// TIA Portal V21 export
TYPE "SafetyPLCSignal"
   STRUCT
      "Circuito sicurezze Ok" : Bool;   // Circuito sicurezza abilitato
      "Circuito sicurezze Ritardate Ok" : Bool;   // Circuito sicurezza ritardato abilitato
      "Richiesta di reset" : Bool;   // Richiesta reset Circuito sicurezza
      "Errore FBK" : Bool;   // Errore Feedback circuito sicurezza
   END_STRUCT;
END_TYPE
